// TIA Portal V17 export
// export: Created 2025-06-26T06:49:23.2699405Z, ExportSetting WithDefaults, DisplayName Totally Integrated Automation Portal, DisplayVersion V17 Update 8, DisplayName TIA Portal Openness, DisplayVersion V17 Update 8, DisplayName TIA Portal Version Control Interface, DisplayVersion V17, DisplayName STEP 7 Professional, DisplayVersion V17 Update 8, DisplayName STEP 7 Safety, DisplayVersion V17 Update 6, DisplayName WinCC Advanced, DisplayVersion V17 Update 8
DATA_BLOCK "InputProcessing_DB"   // DB47
AUTHOR : Heaten
VERSION : 0.1
// stored: AutoNumber true, DBAccessibleFromOPCUA true, DBAccessibleFromWebserver true, InstanceOfName InputProcessing, InstanceOfType FB
"InputProcessing"
   // VAR
   //    AnalogInputProcessing_DB { ExternalAccessible := 'False'; ExternalVisible := 'False'; ExternalWritable := 'False'} : "AnalogInputProcessing";
   //    InputAlarmHandling_DB { ExternalAccessible := 'False'; ExternalVisible := 'False'; ExternalWritable := 'False'} : "InputAlarmHandling";
   //    InverterDriveProcessing_DB : "InverterDriveProcessing";
   //    DigitalInputProcessing_DB { ExternalAccessible := 'False'; ExternalVisible := 'False'; ExternalWritable := 'False'} : "DigitalInputProcessing";
   //    Simulation_DB { ExternalAccessible := 'False'; ExternalVisible := 'False'; ExternalWritable := 'False'} : "Simulation";
   //    HBL_HV_640 { S7_SetPoint := 'True'} : "fbProcessValve2_V2";
   //    HBL_HV_670 { S7_SetPoint := 'True'} : "fbProcessValve2_V2";
   //    CPC_HV_852 { S7_SetPoint := 'True'} : "fbProcessValve2_V2";
   //    HBL_HV_861 { S7_SetPoint := 'True'} : "fbProcessValve2_V2";
   //    bTempOpenReq { S7_SetPoint := 'True'} : Bool;
   //    bTempCloseReq : Bool;
   //    bTempOpenStat : Bool;
   //    bTempCloseStat : Bool;
   // END_VAR
BEGIN
END_DATA_BLOCK
